// TIA Portal V18 export
VAR_GLOBAL   // PLC tag table "DI"
   "H/SSR_019_XV01_OPENFB" AT %I7.4 : Bool;
   "H/SSR_019_XV01_CLOSEFB" AT %I7.5 : Bool;
   "H/SSR_019_XV02_OPENFB" AT %I7.6 : Bool;
   "H/SSR_019_XV02_CLOSEFB" AT %I7.7 : Bool;
   "H/SSR_019_XV03_OPENFB" AT %I8.0 : Bool;
   "H/SSR_019_XV03_CLOSEFB" AT %I8.1 : Bool;
   "H/SSR_019_XV04_CLOSEFB" AT %I8.2 : Bool;
   "H/SSR_019_XV04_OPENFB" AT %I8.3 : Bool;
   "H/SSR_019_XV05_OPENFB" AT %I8.4 : Bool;
   "H/SSR_019_XV05_CLOSEFB" AT %I8.5 : Bool;
   "H/SSR_019_XV06_OPENFB" AT %I8.6 : Bool;
   "H/SSR_019_XV06_CLOSEFB" AT %I8.7 : Bool;
   "H/SSR_019_XV07_OPENFB" AT %I9.0 : Bool;
   "H/SSR_019_XV07_CLOSEFB" AT %I9.1 : Bool;
   "H/SSR_019_XV08_OPENFB" AT %I9.2 : Bool;
   "H/SSR_019_XV08_CLOSEFB" AT %I9.3 : Bool;
   "H/SSR_019_XV09_OPENFB" AT %I9.4 : Bool;
   "H/SSR_019_XV09_CLOSEFB" AT %I9.5 : Bool;
   "H/SSR_019_XV10_OPENFB" AT %I9.6 : Bool;
   "H/SSR_019_XV10_CLOSEFB" AT %I9.7 : Bool;
   "H/SSR_019_XV11_OPENFB" AT %I10.0 : Bool;
   "H/SSR_019_XV11_CLOSEFB" AT %I10.1 : Bool;
   "H/SSR_019_XV12_OPENFB" AT %I10.2 : Bool;
   "H/SSR_019_XV12_CLOSEFB" AT %I10.3 : Bool;
   "H/SSR_019_XV13_OPENFB" AT %I10.4 : Bool;
   "H/SSR_019_XV13_CLOSEFB" AT %I10.5 : Bool;
   "H/SSR_019_AG_RUNFB" AT %I10.6 : Bool;
   "H/SSR_019_AG_STOPFB" AT %I10.7 : Bool;
   "H/SSR_019_AG_TRIP" AT %I11.0 : Bool;
END_VAR
